Fanuc KAREL source: kx00032.KL

-- PROVISIONAL review KL for V1013-1; original PC SHA256 56e39bf5dcc02d1b87d4d41bd6290b1bcd423dd61ded855107d3a2762544b579
-- Incomplete behavior may be omitted. Consult companion uncertainty JSON. Do not deploy.
PROGRAM KX00032
%NOLOCKGROUP
VAR
  I : INTEGER
  J : INTEGER
  B : BOOLEAN
  F : FILE
  S : STRING[80]
-- UNRESOLVED_DECL P type=000102
BEGIN
  -- UNRESOLVED_PC offsets 5-12; opcodes 9D,23
  -- UNRESOLVED_PC offsets 17-21; opcodes 7F
END KX00032
